{attribute addProperty BoxType "KL6581-0002"}
{attribute addProperty Id "StatusAT %I*USINT000Input_CNODEAT %I*USINT000Input_ORGAT %I*USINT000Input_DB0AT %I*USINT000Input_DB1AT %I*USINT000Input_DB2AT %I*USINT000Input_DB3AT %I*USINT000Input_ID0AT %I*USINT000Input_ID1AT %I*USINT000Input_ID2AT %I*USINT000Input_ID3AT %I*USINT000Input_STATUSAT %I*USINT000ControlAT %Q*USINT000Output_CNODEAT %Q*USINT000Output_ORGAT %Q*USINT000Output_DB0AT %Q*USINT000Output_DB1AT %Q*USINT000Output_DB2AT %Q*USINT000Output_DB3AT %Q*USINT000Output_ID0AT %Q*USINT000Output_ID1AT %Q*USINT000Output_ID2AT %Q*USINT000Output_ID3AT %Q*USINT000Output_STATUSAT %Q*USINT000"}
{attribute addProperty CRC "1664645721"}
{attribute addProperty SizeInBites "0"}
{attribute addProperty SizeInBytes "0"}
TYPE Channel_63387A59 :
STRUCT
	{attribute addProperty Name "Status"}
	Status AT %I* : USINT;
	{attribute addProperty Name "Input_CNODE"}
	Input_CNODE AT %I* : USINT;
	{attribute addProperty Name "Input_ORG"}
	Input_ORG AT %I* : USINT;
	{attribute addProperty Name "Input_DB0"}
	Input_DB0 AT %I* : USINT;
	{attribute addProperty Name "Input_DB1"}
	Input_DB1 AT %I* : USINT;
	{attribute addProperty Name "Input_DB2"}
	Input_DB2 AT %I* : USINT;
	{attribute addProperty Name "Input_DB3"}
	Input_DB3 AT %I* : USINT;
	{attribute addProperty Name "Input_ID0"}
	Input_ID0 AT %I* : USINT;
	{attribute addProperty Name "Input_ID1"}
	Input_ID1 AT %I* : USINT;
	{attribute addProperty Name "Input_ID2"}
	Input_ID2 AT %I* : USINT;
	{attribute addProperty Name "Input_ID3"}
	Input_ID3 AT %I* : USINT;
	{attribute addProperty Name "Input_STATUS"}
	Input_STATUS AT %I* : USINT;
	{attribute addProperty Name "Control"}
	Control AT %Q* : USINT;
	{attribute addProperty Name "Output_CNODE"}
	Output_CNODE AT %Q* : USINT;
	{attribute addProperty Name "Output_ORG"}
	Output_ORG AT %Q* : USINT;
	{attribute addProperty Name "Output_DB0"}
	Output_DB0 AT %Q* : USINT;
	{attribute addProperty Name "Output_DB1"}
	Output_DB1 AT %Q* : USINT;
	{attribute addProperty Name "Output_DB2"}
	Output_DB2 AT %Q* : USINT;
	{attribute addProperty Name "Output_DB3"}
	Output_DB3 AT %Q* : USINT;
	{attribute addProperty Name "Output_ID0"}
	Output_ID0 AT %Q* : USINT;
	{attribute addProperty Name "Output_ID1"}
	Output_ID1 AT %Q* : USINT;
	{attribute addProperty Name "Output_ID2"}
	Output_ID2 AT %Q* : USINT;
	{attribute addProperty Name "Output_ID3"}
	Output_ID3 AT %Q* : USINT;
	{attribute addProperty Name "Output_STATUS"}
	Output_STATUS AT %Q* : USINT;
END_STRUCT
END_TYPE

(* stored: Version 1.2.0.0, ProductVersion 3.1.4024.9
   DUT Channel_63387A59: Id {e835ce8a-b8a7-442f-860d-f92abd5e3c3e} *)
